Fanuc KAREL source: IO0021.compact.KL

PROGRAM IO0021
%STACKSIZE=65535
%PRIORITY=65535
%NOLOCKGROUP
ROUTINE RTEST FROM IO0021
ROUTINE RTEST
VAR
L1 : ARRAY[3] OF INTEGER
L2 : XYZWPR
L3 : JOINTPOS9
L4 : POSITION
S1 : INTEGER
U2C_38 : REAL
U2C_39 : REAL
U2C_40 : BOOLEAN
U2C_41 : REAL
BEGIN
S1=1
L1[1]=2
U2C_40=TRUE
U2C_41=1.0
IF (DOUT[17]=TRUE) THEN
S1=(S1 + 1)
ENDIF
END RTEST
BEGIN
RTEST
END IO0021
